{attribute 'reflection'}
FUNCTION_BLOCK PUBLIC FB_DevAnalogInAutoCalibrate EXTENDS FB_DevAnalogInputScaled
VAR_INPUT
END_VAR
VAR_OUTPUT
END_VAR
VAR
END_VAR

SUPER^(refFbFault := refFbFault);

METHOD PUBLIC CmdCalibrateNull : BOOL
VAR_INPUT
END_VAR
// set offset to calibrate to null
nOfset := - inHwInput ;
END_METHOD

METHOD PUBLIC CmdCalilbrateValue : BOOL // calibrate gain factor to actual value (warning calibrate to null before calibrating to value)
VAR_INPUT
	fCalibrationValue	: LREAL ; // Active input value to sensor (calibration setpoint)
END_VAR
// set gain from current value
fGainFactor := INT_TO_LREAL(inHwInput + nOfset) / fCalibrationValue ;
END_METHOD

END_FUNCTION_BLOCK

(* stored: Version 1.1.0.1, ProductVersion 3.1.4024.5
   POU FB_DevAnalogInAutoCalibrate: Id {52f8b1c3-b2bf-0db6-00eb-320245a39b92}, SpecialFunc None
   Method CmdCalibrateNull: Id {dc1e7d0d-643f-0785-3788-917d8619bf0a}
   Method CmdCalilbrateValue: Id {a5144a45-d837-0a3b-1129-ae07bd4b6a95} *)
